RoboDK station: project.rdk

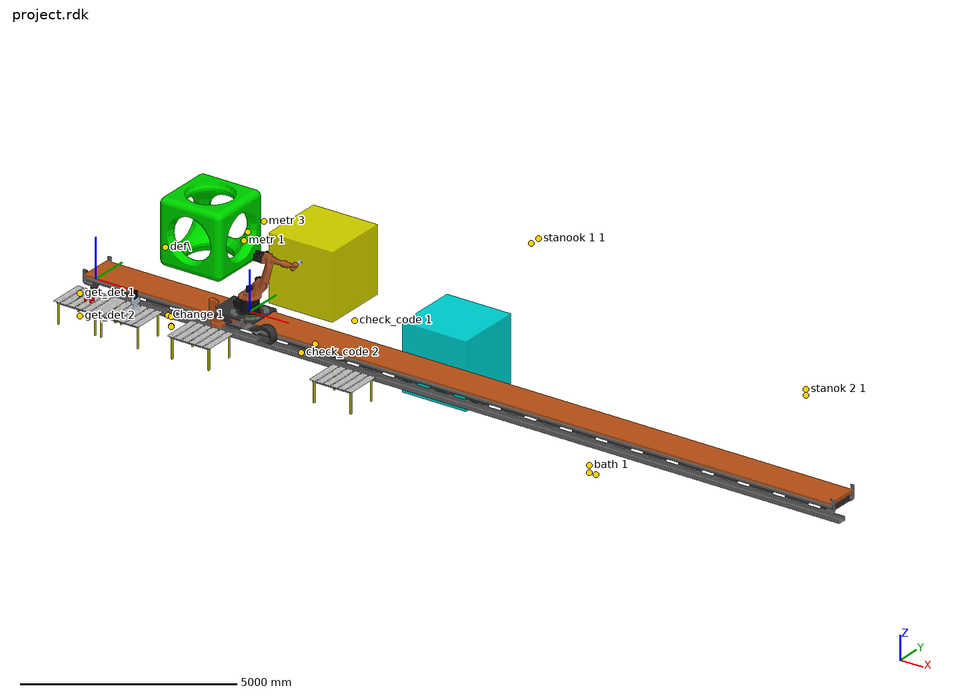
[picture v0: the station drawn from its stored meshes, robots at their saved joint values, targets as dots, program paths as lines]
Station project. Poses are relative to the parent item; angles as X-Y-Z fixed-axis rotations.
  - frame ABB IRBT 6004 Standard 20m Base at (0, 2000, 0) mm
    - robot Platform: 1 axes, repeatability 0.1 mm
        modified DH rows (alpha deg, a mm, theta deg, d mm): 0, 0, 0, 0 linear
        base shift (840.5, 4.2, 379.5) mm, rotated rx 0 ry 90 rz 0 deg
        joint limits [0] to [20000]; home [0]; saved at [3500]
      - frame KUKA KR 16 2 Base at (0, 0, 0) mm
        - robot Robot: 6 axes, payload 16 kg, reach 901 mm, repeatability 0.05 mm, weight 235 kg
            modified DH rows (alpha deg, a mm, theta deg, d mm): 0, 0, 0, 675; -90, 260, 0, 0; 0, 680, -90, 0; -90, -35, 0, 670; 90, 0, 0, 0; -90, 0, 180, 158
            joint limits [-185, -155, -130, -350, -130, -350] to [185, 35, 154, 350, 130, 350]; home [0, -90, 90, 0, 0, 0]; saved at [-48.922, -74.781, 98.374, -112.776, 45.747, 124.401]
          - tool Gripper, TCP at (0, 0, 233.37) mm, size 100 x 89.2 x 240.5 mm
    - target def\ (Cartesian target) at (1966.18, 4.2, 1360.56) mm, rotated rx -150 ry 0 rz -90 deg; joints [0, -90, 90, 0, 60, 90, 0] of Robot
    - object Pallet at (800, -1500, 300) mm, size 1193.8 x 965.2 x 609.6 mm, geometry from Object Table.wrl
      - object Part1 at (50, 0, 50) mm, size 60 x 60 x 80 mm, geometry from part.sld
      - object Part2 at (190, 0, 50) mm, size 60 x 60 x 80 mm, geometry from part.sld
      - object Part3 at (50, -120, 50) mm, size 60 x 60 x 80 mm
      - object Part4 at (190, -120, 50) mm, size 60 x 60 x 80 mm, geometry from part.sld
      - target get_det 1 (Cartesian target) at (850, -1500, 1000) mm, rotated rx 180 ry 0 rz -180 deg; joints [89.638, -32.439, 31.83, 0, 90.609, 89.638, 0] of Robot
      - target get_det 2 (Cartesian target) at (850, -1500, 403.49) mm, rotated rx 180 ry 0 rz 180 deg; joints [89.638, -7.877, 36.615, 180, -61.262, -90.362, 0] of Robot
    - object Check at (4000, -1500, 300) mm, size 1193.8 x 965.2 x 609.6 mm, geometry from Object Table.wrl
      - target check_code 1 (Cartesian target) at (4349.5, 4.2, 1562.67) mm, rotated rx -150 ry 0 rz -90 deg; joints [0, -98.007, 80.008, 0, 77.998, 90, 2500] of Robot
      - target check_code 2 (Cartesian target) at (3982.35, -1626.73, 1284.65) mm, rotated rx -93.64 ry 4.54 rz 178.33 deg; joints [70.009, -49.435, 69.401, -234.657, 26.481, -44.352, 2700] of Robot
      - target check_code 3 (Cartesian target) at (4029.8, -1122.76, 1320.04) mm, rotated rx 150 ry -68.14 rz -55.12 deg; joints [48.492, -78.25, 99.365, 86.7, 36.186, 91.037, 2500] of Robot
    - object Change at (2000, -1500, 300) mm, size 1193.8 x 965.2 x 609.6 mm, geometry from Object Table.wrl
      - object Gripper at (32.23, 204.34, 7.59) mm, rotated rx 0 ry 0 rz 90 deg, size 200 x 178.4 x 481.1 mm
      - target Change 1 (Cartesian target) at (2000, -1300, 1000) mm, rotated rx -180 ry 0 rz -180 deg; joints [91.779, -53.241, 68.304, 0, 74.937, 91.779, 1200] of Robot
      - target Change 2 (Cartesian target) at (2100, -1300, 1000) mm, rotated rx 180 ry 0 rz 90 deg; joints [87.388, -53.179, 68.203, 0, 74.976, -2.612, 1200] of Robot
      - target Change 3 (Cartesian target) at (2100, -1300, 760) mm, rotated rx 180 ry 0 rz 90 deg; joints [87.388, -43.97, 74.988, 0, 58.983, -2.612, 1200] of Robot
      - target Change 4 (Cartesian target) at (2100, -1300, 750) mm, rotated rx 0 ry -90 rz 0 deg; joints [70.929, -15.343, 58.576, 76.678, 103.771, 45.151, 1200] of Robot
    - object Bath at (8000, -1500, 300) mm, size 1193.8 x 965.2 x 609.6 mm, geometry from Object Table.wrl
      - target bath 1 (Cartesian target) at (8000, -1500, 600) mm, rotated rx 180 ry 0 rz -180 deg; joints [91.542, -19.628, 42.394, 0, 67.234, 91.542, 7200] of Robot
      - target bath 2 (Cartesian target) at (8000, -1500, 400) mm, rotated rx -180 ry 0 rz 180 deg; joints [91.542, -7.575, 36.308, 0, 61.267, 91.542, 7200] of Robot
      - target bath 3 (Cartesian target) at (8200, -1500, 400) mm, rotated rx -180 ry 0 rz -180 deg; joints [83.947, -6.658, 34.312, 0, 62.346, 83.947, 7200] of Robot
    - object Stan_1 at (5000, 2000, 1000) mm, size 1800 x 1800 x 1800 mm, geometry from box.sld
      - target stanook 1 1 (Cartesian target) at (5000, 1535.02, 1420) mm, rotated rx 0 ry 90 rz 90 deg; joints [-59.938, -52.972, 65.311, -110.265, 32.275, 113.591, 3500] of Robot
      - target stanook 1 2 (Cartesian target) at (5000, 1250, 1420) mm, rotated rx 0 ry 90 rz 90 deg; joints [-52.337, -71.994, 93.782, -115.683, 42.687, 123.194, 3500] of Robot
    - object Stan_2 at (8900, 1800, -120) mm, size 1800 x 1800 x 1800 mm, geometry from box.sld
      - target stanok 2 1 (Cartesian target) at (9000, 1200, 1100) mm, rotated rx 180 ry 0 rz -90 deg; joints [-91.94, -64.784, 77.208, 0, 77.576, -1.94, 8200] of Robot
      - target stanok 2 2 (Cartesian target) at (9000, 1200, 941.44) mm, rotated rx 180 ry 0 rz -90 deg; joints [-91.94, -59.866, 84.376, 0, 65.49, -1.94, 8200] of Robot
    - object Stan_3 at (1000, 1000, 200) mm, size 1749.9 x 1749.9 x 1749.9 mm, geometry from Box.stl
      - target metr 1 (Cartesian target) at (2466.18, 4.2, 1360.56) mm, rotated rx -150 ry 0 rz -90 deg; joints [0, -90, 90, 0, 60, 90, 500] of Robot
      - target metr 2 (Cartesian target) at (2100.11, 699.99, 1199.94) mm, rotated rx -90 ry 0 rz 0 deg; joints [-21.839, -78.504, 126.448, -106.571, 75.571, 230.057, 500] of Robot
      - target metr 3 (Cartesian target) at (2100.11, 1356.42, 1199.94) mm, rotated rx -90 ry 0 rz 0 deg; joints [-51.671, -51.961, 84.526, -124.249, 48.613, 225.841, 500] of Robot
